INTERFACE ITF_AxisStatus EXTENDS __SYSTEM.IQueryInterface

METHOD getCurrentPosition : LREAL
VAR_INPUT
END_VAR
END_METHOD

METHOD HasError : BOOL
VAR_INPUT
END_VAR
END_METHOD

METHOD isAtPosition : BOOL
VAR_INPUT
	position : MC_LREAL;
END_VAR
END_METHOD

METHOD isEnabled : BOOL
VAR_INPUT
END_VAR
END_METHOD

METHOD isStationary : BOOL
VAR_INPUT
END_VAR
END_METHOD

END_INTERFACE

(* stored: Version 1.1.0.1
   Itf ITF_AxisStatus: Id {6057db56-1d8d-4c90-8f15-4379a266ab62}
   Method getCurrentPosition: Id {4fa41b0c-b611-436e-9bd7-2a6e55e87dc6}
   Method HasError: Id {e7471b4a-08a6-46c7-9890-534c8ede1daa}
   Method isAtPosition: Id {b1b2fe74-f8e0-4241-b0e9-3e1b63b14a12}
   Method isEnabled: Id {206658e1-36fc-414b-a92b-edd9aceba017}
   Method isStationary: Id {58e66eb5-9088-44a9-a122-982f73f5789e} *)
